KUKA KRL program: FORCE_X.src, FORCE_X.dat

--- FORCE_X.src ---
&ACCESS RVP
&REL 74
&PARAM TEMPLATE = C:\KRC\Roboter\Template\vorgabe
&PARAM EDITMASK = *
DEF FORCE_X( )
INT X

DECL BOOL TEMP
DECL BOOL HEMP
DECL BOOL SEMP
DECL FRAME SETPNT
DECL FRAME PT, PT2
DECL CHAR X1
DECL INT NUM

X1="Y"

;FOLD INI
  ;FOLD BASISTECH INI
    GLOBAL INTERRUPT DECL 3 WHEN $STOPMESS==TRUE DO IR_STOPM ( )
    INTERRUPT ON 3
    BAS (#INITMOV,0 )
  ;ENDFOLD (BASISTECH INI)
  ;FOLD USER INI
    ;Make your modifications here

  ;ENDFOLD (USER INI)
;ENDFOLD (INI)

$STIFFNESS.STRATEGY=10
$STIFFNESS.COMMIT=TRUE
$OV_PRO=75
$ORI_TYPE=#CONSTANT
$TOOL=TOOL_DATA[5]

FOR X=1 TO 6
$ACC_AXIS[X]=70
$VEL_AXIS[X]=70
ENDFOR


;FOLD PTP PT3 Vel=100 % PDAT3 Tool[5]:Pneumatic_gripper_probe Base[0];%{PE}%R 5.6.11,%MKUKATPBASIS,%CMOVE,%VPTP,%P 1:PTP, 2:PT3, 3:, 5:100, 7:PDAT3
$BWDSTART=FALSE
PDAT_ACT=PPDAT3
FDAT_ACT=FPT3
BAS(#PTP_PARAMS,100)
PTP XPT3
;ENDFOLD

PT2= GETPOINT(X1,1)
PTP PT2

LIN_REL{Z -30}

TEMP=TRIGX()
HEMP=SOFTINY()
SEMP=FORCEY()

LIN_REL {Y 5}

HALT

$STIFFNESS.STRATEGY=10
$STIFFNESS.COMMIT=TRUE
$OV_PRO=50

;FOLD PTP HOME  Vel= 100 % DEFAULT;%{PE}%MKUKATPBASIS,%CMOVE,%VPTP,%P 1:PTP, 2:HOME, 3:, 5:100, 7:DEFAULT
$BWDSTART = FALSE
PDAT_ACT=PDEFAULT
FDAT_ACT=FHOME
BAS (#PTP_PARAMS,100 )
$H_POS=XHOME
PTP  XHOME
;ENDFOLD


END

--- FORCE_X.dat ---
&ACCESS RVP
&REL 74
&PARAM TEMPLATE = C:\KRC\Roboter\Template\vorgabe
&PARAM EDITMASK = *
DEFDAT  FORCE_X
;FOLD EXTERNAL DECLARATIONS;%{PE}%MKUKATPBASIS,%CEXT,%VCOMMON,%P
;FOLD BASISTECH EXT;%{PE}%MKUKATPBASIS,%CEXT,%VEXT,%P
EXT  BAS (BAS_COMMAND  :IN,REAL  :IN )
DECL INT SUCCESS
;ENDFOLD (BASISTECH EXT)
;FOLD USER EXT;%{E}%MKUKATPUSER,%CEXT,%VEXT,%P
;Make here your modifications

;ENDFOLD (USER EXT)
;ENDFOLD (EXTERNAL DECLARATIONS)
DECL BASIS_SUGG_T LAST_BASIS={POINT1[] "HOME                    ",POINT2[] "HOME                    ",CP_PARAMS[] "CPDAT0                  ",PTP_PARAMS[] "PDAT3                   ",CONT[] "                        ",CP_VEL[] "2.0                     ",PTP_VEL[] "100                     ",SYNC_PARAMS[] "SYNCDAT                 ",SPL_NAME[] "S0                      "}
DECL E6POS XP1={X -25.6887207,Y -592.06842,Z 79.8191605,A 0.0109860497,B 0.00211965106,C -179.962494,S 1,T 44,E1 0.000214576707,E2 0.0,E3 0.0,E4 0.0,E5 0.0,E6 0.0}
DECL FDAT FP1={TOOL_NO 5,BASE_NO 0,IPO_FRAME #BASE,POINT2[] " ",TQ_STATE FALSE}
DECL PDAT PPDAT1={VEL 100.0,ACC 100.0,APO_DIST 100.0,APO_MODE #CPTP}
DECL E6POS XP2={X -25.6882095,Y -592.078918,Z 46.9154587,A 0.0110969897,B 0.00197515101,C -179.964493,S 1,T 44,E1 0.000291824312,E2 0.0,E3 0.0,E4 0.0,E5 0.0,E6 0.0}
DECL FDAT FP2={TOOL_NO 5,BASE_NO 0,IPO_FRAME #BASE,POINT2[] " ",TQ_STATE FALSE}
DECL PDAT PPDAT2={VEL 100.0,ACC 100.0,APO_DIST 100.0,APO_MODE #CPTP}
DECL PDAT PPDAT3={VEL 100.0,ACC 100.0,APO_DIST 100.0,APO_MODE #CPTP}
DECL E6POS XPT3={X 12.2777205,Y -591.623108,Z 336.000305,A 1.18348396,B -0.000385531195,C -179.988007,S 1,T 36,E1 -0.0136213303,E2 0.0,E3 0.0,E4 0.0,E5 0.0,E6 0.0}
DECL FDAT FPT3={TOOL_NO 5,BASE_NO 0,IPO_FRAME #BASE,POINT2[] " ",TQ_STATE FALSE}
ENDDAT
